TEXTLIST PDVConfigMode
  0 = 'No C'
  1 = 'ZERO'
  2 = 'Pre.Alig'
   = ''
END_TEXTLIST

(* stored: Version 1.1.0.1, ProductVersion 3.1.4024.4
   TextList PDVConfigMode: Id {6919b340-ee1b-489c-9a26-bcd2629a042d} *)
